TYPE Cnv_Instruction_DUT :
STRUCT
	Mode_Change:	UINT;
	Stop:	BOOL;
	Enable:	BOOL;
	Reset:	BOOL;
	Execute:	BOOL;
	Task_ID:	UINT;
	Task_Metadata:	STRING;
	Transfer_To_ID:	DINT;
	Transfer_From_ID:	DINT;
	Transfer_in_Progress:	BOOL;
	Inbound_Ready:	BOOL;
	Transfer_Complete:	BOOL;
	Outbound_Ready:	BOOL;
	Start_Transfer:	BOOL;
	Foward:	BOOL;
	Backward:	BOOL;
END_STRUCT
END_TYPE

(* stored: Version 1.1.0.1
   DUT Cnv_Instruction_DUT: Id {fb11704c-2120-49a6-b539-5bf67c9015dd} *)
